// TIA Portal V20 export
TYPE "Rollerbed_Configuration"
   STRUCT
      StopDetSetUsed : Bool;
      LowSpeedDetSetUsed : Bool;
      LSpeedDetSetConstOn : Bool;
      TrainActivatedSet : Bool;
      TrfInSetUsed : Bool;
      TrfOutSetUsed : Bool;
      TrspNoLowSpeed : Bool;
      InitDirection : Bool;
      RevSwUsed : Bool;
      StopDetResUsed : Bool;
      LowSpeedDetResUsed : Bool;
      LSpeedDetResConstOn : Bool;
      TrainActivatedRes : Bool;
      TrfInResUsed : Bool;
      TrfOutResUsed : Bool;
      SafetySwNc : Bool;
      SafetySwUsed : Bool;
      ReleaseBrakeUsed : Bool;
      MotorProtectionSwNc : Bool;
      MotorProtectionUsed : Bool;
   END_STRUCT;
END_TYPE
